FUNCTION F_FUN : BOOL
VAR_INPUT
END_VAR
VAR
	var1			: __SYSTEM.VAR_INFO;
	var2			: __SYSTEM.VAR_INFO;
	fbLog			: FB_Logger('F_FUN (Inst)');
END_VAR
VAR_STAT
	fbLog2			: FB_Logger('F_FUN (Stat)');
END_VAR

fbLog();
fbLog2();
var1 := __VARINFO(fbLog);
var2 := __VARINFO(fbLog2);

END_FUNCTION

(* stored: Version 1.1.0.1, ProductVersion 3.1.4024.0
   POU F_FUN: Id {66f1fd3f-30bd-4766-a4ba-288de1fa6c2c}, SpecialFunc None *)
